// LS Electric XG5000 project: PROJECT_1
// PLC LSPLC

PROGRAM InverterCom (task: 스캔 프로그램)

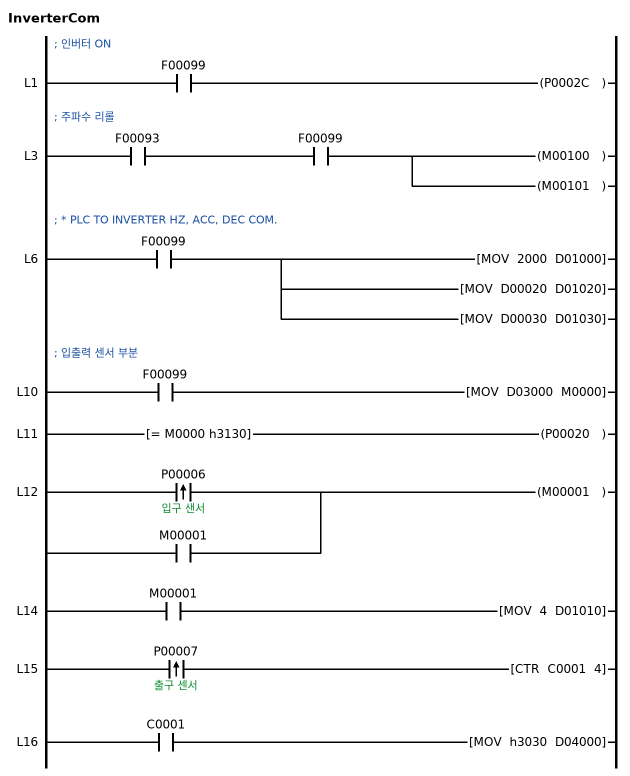
// 인버터 ON
; L1
LOAD      F00099
OUT       P0002C
// 주파수 리롤
; L3
LOAD      F00093
AND       F00099
OUT       M00100
OUT       M00101
// * PLC TO INVERTER HZ, ACC, DEC COM.
; L6
LOAD      F00099
MOV       2000 D01000
MOV       D00020 D01020
MOV       D00030 D01030
// 입출력 센서 부분
; L10
LOAD      F00099
MOV       D03000 M0000
; L11
LOAD=     M0000 h3130
OUT       P00020
; L12
LOADP     P00006	// 입구 샌서
OR        M00001
OUT       M00001
; L14
LOAD      M00001
MOV       4 D01010
; L15
LOADP     P00007	// 출구 센서
CTR       C0001 4
; L16
LOAD      C0001
MOV       h3030 D04000
// * INVETER MANUAL OPERATION